(* IEC 61131-3 sources: PUA/, 3 files *)

(* ---- Types.typ ---- *)
TYPE
	RoomTyp : STRUCT
		diPstryk : ARRAY[1..2] OF BOOL; (* Obsługa włączników światła *)
		doLampa : ARRAY[1..2] OF BOOL; (* obsługa lamp *)
		diTemperatura : INT; (* Odczyt Temperatury - sonda PT1000 *)
		diFotokomorka : ARRAY[1..2] OF BOOL; (*Odczyt stygnałów z gotokomorek *)

	END_STRUCT;

	HouseTyp : STRUCT
		Jadalnia : RoomTyp;
		Kuchnia : RoomTyp;
		Sypialnia : RoomTyp;
		Korytarz : RoomTyp;
	END_STRUCT;
END_TYPE

(* ---- Main.st ---- *)
PROGRAM _INIT
	(* Insert code here *)
	uiLightControlMode := 5; //case 5
	//uiZegar_PT[1] := 1
	(* ALE NIE WIEM CZY PONIZSZE USTAWIENIA DZIALAJA *)
	uiZegarTON_PT[1] := 1;
	//ZegarTON[2].PT := 3;
	uiZegarTON_PT[2] := 3;
	uiZegarTOF_PT[1] := 3;

END_PROGRAM

PROGRAM _CYCLIC
	(* Insert code here *)
	CASE uiLightControlMode OF
		1: //Klasyczne sterowanie z włącznikimem bistabilnym
			Dom.Jadalnia.doLampa[1] := Dom.Jadalnia.diPstryk[1];
		2: //dotyk
			Dom.Jadalnia.doLampa[1] := EDGEPOS(Dom.Jadalnia.diPstryk[1]) XOR Dom.Jadalnia.doLampa[1];
		3: //swiatlo mrugajace
			ZegarTON[1].IN:= Dom.Jadalnia.diPstryk[2] AND NOT(ZegarTON[1].Q);
		//	ZegarTon[1].PT:= T#1s; //zadanie czasu 1s poprzez deklaracje T#
			//ZegarTon[1].PT:= REAL_TO_TIME(uiZegarTON_PT[1]*1000); //zadanie czasu 1s poprzez deklaracje T#

			ZegarTON[1](); //FUB
			Dom.Jadalnia.doLampa[1] := Dom.Jadalnia.diPstryk[2] AND (ZegarTON[1].Q XOR Dom.Jadalnia.doLampa[1]);
			IF EDGEPOS(Dom.Jadalnia.doLampa[1]) THEN
				ZegarTON[1].PT := REAL_TO_TIME(uiZegarTON_PT[1]*1000);
			END_IF
			IF EDGENEG(Dom.Jadalnia.doLampa[1]) THEN
				ZegarTON[1].PT := REAL_TO_TIME(uiZegarTON_PT[2]*1000);
			END_IF
		4:
			ZegarTOF[1].IN := Dom.Korytarz.diFotokomorka[1];
			ZegarTOF[1].PT := REAL_TO_TIME(uiZegarTOF_PT[1] *1000);
			ZegarTOF[1]();
			Dom.Korytarz.doLampa[1] := ZegarTOF[1].Q;
		5: //Ściemniacz\
			//POTENCJOMETR
//			Skaluj[1].x := INT_TO_REAL(Dom.Jadalnia.aiSciemniacz[1]);
//			Skaluj[1].x1 := 0;
//			Skaluj[1].y1 := 13000;
//			Skaluj[1].x2 := 32767;
//			Skaluj[1].y2 := 30000;
//			Skaluj[1]();
			//	Dom.Jadalnia.aoLampa[1] := REAL_TO_INT(Skaluj[1].y);
			//TERMOMETR
			Skaluj[1].x := INT_TO_REAL(Dom.Jadalnia.aiSciemniacz[2]);
			Skaluj[1].x1 := 320; (*dolna temperatura w termometrze *)
			Skaluj[1].y1 := 13000; (*dolna granica w ktorej, zarowka jeszcze nie swieci *)
			Skaluj[1].x2 := 370; (*gorna granica temperatury *)
			Skaluj[1].y2 := 30000; (*gorna granica swiecenia zarowk *)
			Skaluj[1]();
			Dom.Jadalnia.aoLampa[1] := REAL_TO_INT(Skaluj[1].y);

		//Dom.Korytarz.doLampa[1] :=
	END_CASE

END_PROGRAM

PROGRAM _EXIT
	(* Insert code here *)

END_PROGRAM

(* ---- Variables.var ---- *)
VAR
	Dom : HouseTyp;
	uiLightControlMode : USINT; (* tryb pracy oswietlenia : 1 - klasyczne sterowanie, 2- orzycisk dwustanowy, 3 -swiatlo pulsujace ze stalym zboczem, 4 swiatlo pulsujace ze zmiennym zboczem *)
	ZegarTON : ARRAY[1..10] OF TON;
	ZegarTOF : ARRAY[1..10] OF TOF;
	Skaluj : ARRAY[1..10] OF LCRLimScal;
END_VAR

VAR RETAIN (*retain podtrzymuje w pamieci zmienna *)
	uiZegarTON_PT : ARRAY[1..10] OF REAL; (*Czas zadany w sekundach *)
	uiZegarTOF_PT : ARRAY[1..10] OF REAL; (*Czas zadany w sekundach *)
END_VAR
